PROGRAM MAIN
VAR
	PowerLeftWheel		 : MC_Power;
	PowerRightWheel		 : MC_Power;
	LeftWheel			 : AXIS_REF;
	RightWheel			 : AXIS_REF;
	NavitrolInControl	 : BOOL := TRUE;
	StreamVeloLeftWheel	 : FB_StreamVelocity;
	StreamVeloRightWheel : FB_StreamVelocity;
	Supervisor			 : FB_Supervisor := (RemoteHost := '127.0.0.1', RemotePort := 2000);
END_VAR

Supervisor.st1016_Measurement_update_differential_drive.Odometry_left_wheel	 := TO_UDINT(LeftWheel.NcToPlc.ActPos * 10_000_000);
Supervisor.st1016_Measurement_update_differential_drive.Odometry_Right_wheel := TO_UDINT(RightWheel.NcToPlc.ActPos * 10_000_000);
Supervisor(Execute := TRUE);
PowerLeftWheel(Axis			   := LeftWheel,
			   Enable		   := TRUE,
			   Enable_Positive := TRUE,
			   Enable_Negative := TRUE,
			   Override		   := 100.0);

PowerRightWheel(Axis			:= RightWheel,
				Enable			:= TRUE,
				Enable_Positive := TRUE,
				Enable_Negative := TRUE,
				Override		:= 100.0);

StreamVeloLeftWheel(Axis		   := LeftWheel,
					Enable		   := NavitrolInControl,
					TargetVelocity := Supervisor.st1116_Motor_Control_Differential.Speed_Left);

StreamVeloRightWheel(Axis			:= RightWheel,
					 Enable			:= NavitrolInControl,
					 TargetVelocity := Supervisor.st1116_Motor_Control_Differential.Speed_Right);

END_PROGRAM

(* stored: Version 1.1.0.1, ProductVersion 3.1.4026.17
   POU MAIN: Id {3630ccad-c9cd-4213-8e6b-1c2fc4e308ce}, SpecialFunc None *)
